FUNCTION "PL_DigSetValFalse" : Void
{ S7_Optimized_Access := 'TRUE' }
VERSION : 0.1
   VAR_IN_OUT
      In : Byte;
   END_VAR


BEGIN
	#In.%X7 := false;
END_FUNCTION

